{attribute 'qualified_only'}

TYPE camResult :
(
	null          := 0,                         // Неправилен резултат от камерата
	turnCCW,
	turnCW
	
)DINT;
END_TYPE

(* stored: Version 1.1.0.1, ProductVersion 3.1.4024.3
   DUT camResult: Id {540fc52e-1eeb-49ea-a851-71b774fdf73e} *)
